FUNCTION_BLOCK LiftMove (* Basic Function Block Type *)
  (* Standard: 61499-2 *)
  (* Version 0.0, 6/3/2016, Andrei, nxtControl GmbH, Template *)
  PACKAGE Main;
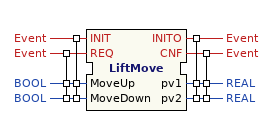
  EVENT_INPUT
    INIT WITH MoveUp, MoveDown; (* Initialization Request *)
    REQ WITH MoveUp, MoveDown; (* Normal Execution Request *)
  END_EVENT
  EVENT_OUTPUT
    INITO WITH pv1, pv2; (* Initialization Confirm *)
    CNF WITH pv1, pv2; (* Execution Confirmation *)
  END_EVENT
  VAR_INPUT
    MoveUp : BOOL; (* Input event qualifier *)
    MoveDown : BOOL;
  END_VAR
  VAR_OUTPUT
    pv1 : REAL; (* Output event qualifier *)
    pv2 : REAL;
  END_VAR
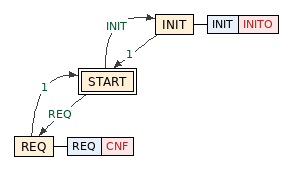
  EC_STATES
    START; (* Initial State *)
    INIT : INIT -> INITO; (* Initialization *)
    REQ : REQ -> CNF; (* Normal execution *)
  END_STATES
  EC_TRANSITIONS
    START TO INIT := INIT;
    INIT TO START := 1;
    START TO REQ := REQ;
    REQ TO START := 1;
  END_TRANSITIONS
  ALGORITHM INIT IN ST: (* Initialization algorithm *)
pv1 := 0.0;
pv2 := 0.0;
  END_ALGORITHM
  ALGORITHM REQ IN ST: (* Normally executed algorithm *)
IF MoveUp AND NOT(MoveDown) THEN
	pv1 := 0.0;
	pv2 := 200.0;
ELSIF MoveDown AND NOT(MoveUp) THEN
	pv1 := 200.0;
	pv2 := 0.0;
ELSE
	pv1 := 0.0;
	pv2 := 0.0;
END_IF;
  END_ALGORITHM
END_FUNCTION_BLOCK
